# EPICS substitutions: db/generated/TOF_PMT.substitutions
# P is supplied by dbLoadTemplate() in st.cmd.
file "db/plsci.template"
{
    pattern
    {
        CHAMBER,PMT
    }

    { FMF2,1 }
    { FMF2,2 }
    { FMF2,3 }
    { FMF2,4 }
    { FMF2,5 }
    { FMF2,6 }
    { FMF2,7 }
    { FMF2,8 }
    { FHF1,1 }
    { FHF1,2 }
    { FHF1,3 }
    { FHF1,4 }
    { FHF1,5 }
    { FHF1,6 }
    { FHF1,7 }
    { FHF1,8 }
}
